// Mitsubishi GX Works2 project: PLC_GROUP_01  (1) (2)   PLC: FX3G

// global labels: Global1
VAR_GLOBAL
  DayStart AT X010 : BOOL;
  DayCoil AT Y010 : BOOL;
  DayEnd AT M0 : BOOL;
  FlourSt AT D1120 : REAL;
  FlourStock AT D1100 : REAL;
  YeastSt AT D1122 : REAL;
  YeastStock AT D1102 : REAL;
  WaterSt AT D1124 : REAL;
  WaterStock AT D1104 : REAL;
  OilSt AT D1126 : REAL;
  OilStock AT D1106 : REAL;
  SpicesSt AT D1128 : REAL;
  SpicesStock AT D1108 : REAL;
  Shutdown AT X007 : BOOL;
  InventoryDone AT M18 : BOOL;
  PrepCoil AT Y005 : BOOL;
END_VAR
VAR_GLOBAL CONSTANT
  Const_100 : REAL := 100;
  Yeast_MUL : REAL := 0.2;
END_VAR
VAR_GLOBAL
  YeastCheck AT D1130 : REAL;
END_VAR
VAR_GLOBAL CONSTANT
  Water_MUL : REAL := 0.5;
END_VAR
VAR_GLOBAL
  WaterCheck AT D1132 : REAL;
END_VAR
VAR_GLOBAL CONSTANT
  Oil_MUL : REAL := 0.3;
END_VAR
VAR_GLOBAL
  OilCheck AT D1134 : REAL;
END_VAR
VAR_GLOBAL CONSTANT
  Spices_MUL : REAL := 0.1;
END_VAR
VAR_GLOBAL
  SpicesCheck AT D1136 : REAL;
  blink2 AT M50 : BOOL;
  TS1 AT M50 : BOOL;
  blinktest AT TS1 : BOOL;
  blink3 AT M52 : BOOL;
  blinktest2 AT TS2 : BOOL;
  blinkA AT TC1 : BOOL;
END_VAR
VAR_GLOBAL CONSTANT
  blinktimems : INT := 5;
END_VAR
VAR_GLOBAL
  blinkB AT TC2 : BOOL;
  EndBlink10 AT CC1 : BOOL;
END_VAR
VAR_GLOBAL CONSTANT
  Count_10 : INT := 6;
END_VAR
VAR_GLOBAL
  EndBlink10_O AT CS1 : BOOL;
  DayCoilchecker AT M20 : BOOL;
  DayEndBlink AT M22 : BOOL;
  PrepStart AT X002 : BOOL;
  PrepT AT TC3 : BOOL;
END_VAR
VAR_GLOBAL CONSTANT
  LightT : INT := 30;
END_VAR
VAR_GLOBAL
  PrepCoilOff AT TS3 : BOOL;
END_VAR
VAR_GLOBAL CONSTANT
  Const_30 : REAL := 30;
  Const_50 : REAL := 50;
  Const_20 : REAL := 20;
  Const_10 : REAL := 10;
END_VAR
VAR_GLOBAL
  TempFlour AT D2000 : REAL;
  TempOil AT D2002 : REAL;
  TempWater AT D2004 : REAL;
  TempYeast AT D2006 : REAL;
  TempSpices AT D2008 : REAL;
  KneadStart AT X001 : BOOL;
  KneadStage AT M30 : BOOL;
  KneadCoil AT Y001 : BOOL;
  MixerStock AT D1110 : REAL;
END_VAR
VAR_GLOBAL CONSTANT
  Const_210 : REAL := 210;
END_VAR
VAR_GLOBAL
  FinishTransfer AT M4 : BOOL;
  Knead AT X011 : BOOL;
  RiseStart AT X011 : BOOL;
  RiseStage AT M40 : BOOL;
  EndBlinkRise AT CS10 : BOOL;
  EndBlinkRise1 AT CC10 : BOOL;
  blinkRise AT M41 : BOOL;
  blinkA_R AT TC10 : BOOL;
  blinkA_R1 AT TS10 : BOOL;
  blinkB_R AT TC11 : BOOL;
  Coil2 AT Y002 : BOOL;
  blinkB_R1 AT TS11 : BOOL;
  Coil3 AT Y003 : BOOL;
  RiseStorage AT D1114 : REAL;
  CountC11 AT CC20 : BOOL;
END_VAR
VAR_GLOBAL CONSTANT
  Count_2 : INT := 2;
END_VAR
VAR_GLOBAL
  CountC11End AT CS20 : BOOL;
  CountC5 AT CC5 : BOOL;
  CountC5End AT CS5 : BOOL;
  RiseSt1 AT M45 : BOOL;
  RiseEnd AT CS10 : BOOL;
  BakeStart AT M60 : BOOL;
  BakingPan AT D1118 : REAL;
  BakeT AT TC14 : BOOL;
END_VAR
VAR_GLOBAL CONSTANT
  LightBakeT : INT := 40;
END_VAR
VAR_GLOBAL
  BakeCoilOff AT TS14 : BOOL;
  BakeCoil AT Y004 : BOOL;
  QA3 AT X003 : BOOL;
END_VAR
VAR_GLOBAL CONSTANT
  Const_1 : REAL := 1;
  Const_5 : REAL := 5;
END_VAR
VAR_GLOBAL
  QA_TRUE AT M80 : BOOL;
  QA_T AT TC15 : BOOL;
END_VAR
VAR_GLOBAL CONSTANT
  LightQAT : INT := 50;
END_VAR
VAR_GLOBAL
  QA_Off AT TS15 : BOOL;
  QACoil AT Y006 : BOOL;
  Shelf AT D3333 : REAL;
  LTAnalogCheck AT M82 : BOOL;
  RST_All AT M100 : BOOL;
  Analog_Moved AT M83 : BOOL;
END_VAR
VAR_GLOBAL CONSTANT
  Const_400 : INT := 400;
  Const_2000 : INT := 2000;
END_VAR
VAR_GLOBAL
  Analog_Value AT D8490 : REAL;
  QA_TRUE2 AT M83 : BOOL;
  Analog_Input_2 AT D8281 : INT;
  RiseMoved AT M61 : BOOL;
  Coil4ON AT M61 : BOOL;
  FlourDone AT M19 : BOOL;
END_VAR

// task Task_01 (event TRUE, interval 0, priority 31): POU_01

PROGRAM POU_01
(* structured ladder/FBD written out as ST: instructions are called as NAME(EN, inputs, outputs); _pN, _eN, _tN stand for wires *)
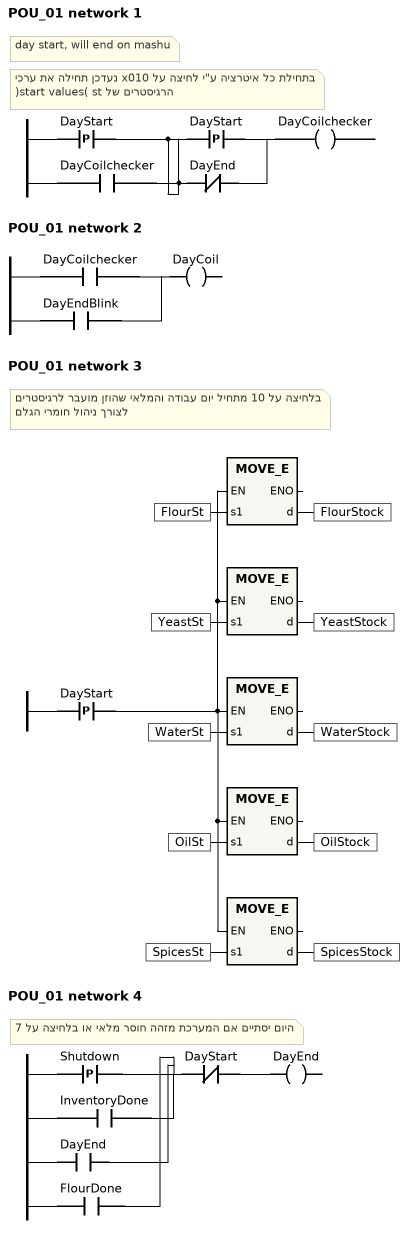
(* network 1 *)
(* day start, will end on mashu *)
(* בתחילת כל איטרציה ע"י לחיצה על x010 נעדכן תחילה את ערכי הרגיסטרים של st )start values( *)
_p1 := LDP(TRUE, DayStart) OR DayCoilchecker;
DayCoilchecker := (_p1 AND LDP(TRUE, DayStart)) OR (_p1 AND NOT DayEnd);
(* network 2 *)
DayCoil := DayCoilchecker OR DayEndBlink;
(* network 3 *)
(* בלחיצה על 10 מתחיל יום עבודה והמלאי שהוזן מועבר לרגיסטרים לצורך ניהול חומרי הגלם *)
_p1 := LDP(TRUE, DayStart);
MOVE_E(_p1, FlourSt, FlourStock);
MOVE_E(_p1, YeastSt, YeastStock);
MOVE_E(_p1, WaterSt, WaterStock);
MOVE_E(_p1, OilSt, OilStock);
MOVE_E(_p1, SpicesSt, SpicesStock);
(* network 4 *)
(* היום יסתיים אם המערכת מזהה חוסר מלאי או בלחיצה על 7 *)
DayEnd := (LDP(TRUE, Shutdown) OR InventoryDone OR DayEnd OR FlourDone) AND NOT DayStart;
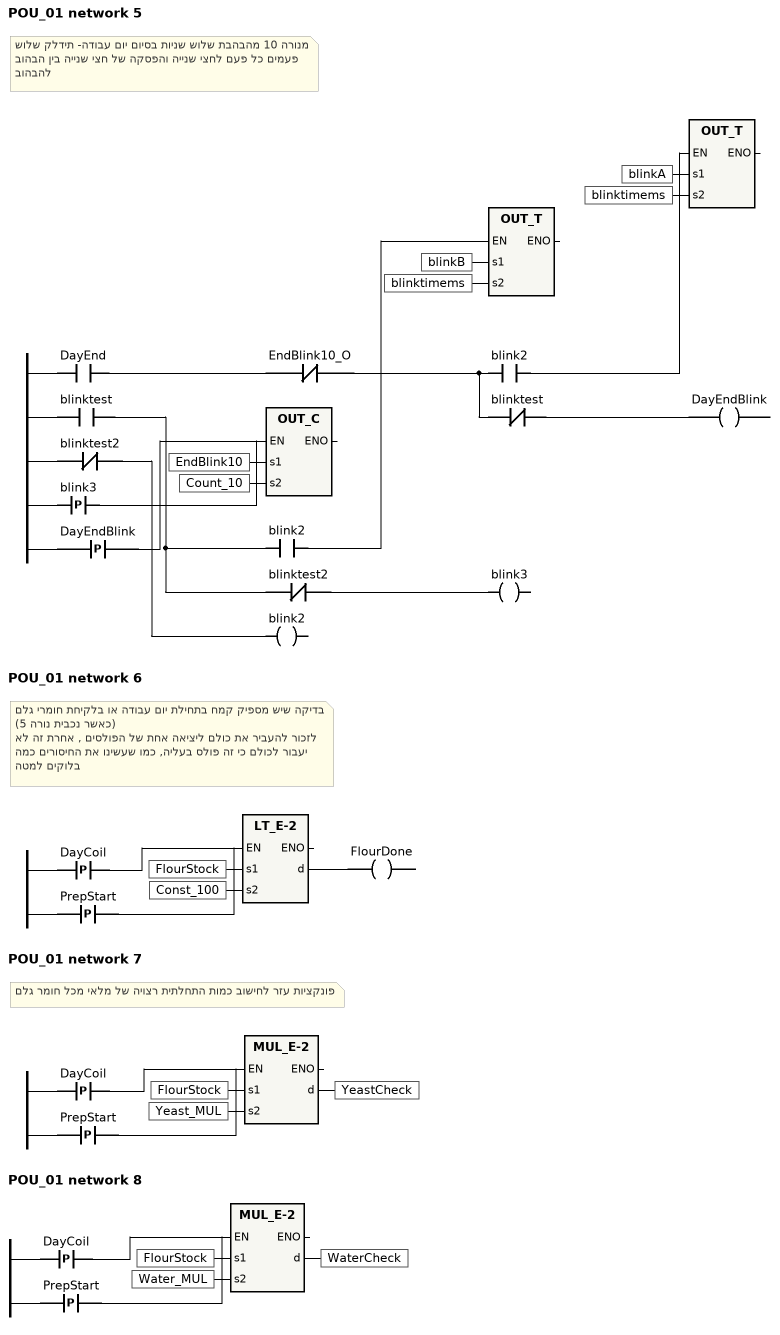
(* network 5 *)
(* מנורה 10 מהבהבת שלוש שניות בסיום יום עבודה- תידלק שלוש פעמים כל פעם לחצי שנייה והפסקה של חצי שנייה בין הבהוב להבהוב *)
_p1 := DayEnd AND NOT EndBlink10_O;
OUT_T(_p1 AND blink2, blinkA, blinktimems);
DayEndBlink := _p1 AND NOT blinktest;
OUT_T(blinktest AND blink2, blinkB, blinktimems);
blink3 := blinktest AND NOT blinktest2;
blink2 := NOT blinktest2;
OUT_C(LDP(TRUE, blink3) OR LDP(TRUE, DayEndBlink), EndBlink10, Count_10);
(* network 6 *)
(* בדיקה שיש מספיק קמח בתחילת יום עבודה או בלקיחת חומרי גלם (כאשר נכבית נורה 5)                                                            לזכור להעביר את כולם ליציאה אחת של הפולסים , אחרת זה לא יעבור לכולם כי זה פולס בעליה, כמו שעשינו את החיסורים כמה בלוקים למטה *)
LT_E(LDP(TRUE, DayCoil) OR LDP(TRUE, PrepStart), FlourStock, Const_100, _t1);
FlourDone := _t1;
(* network 7 *)
(* פונקציות עזר לחישוב כמות התחלתית רצויה של מלאי מכל חומר גלם *)
MUL_E(LDP(TRUE, DayCoil) OR LDP(TRUE, PrepStart), FlourStock, Yeast_MUL, YeastCheck);
(* network 8 *)
MUL_E(LDP(TRUE, DayCoil) OR LDP(TRUE, PrepStart), FlourStock, Water_MUL, WaterCheck);
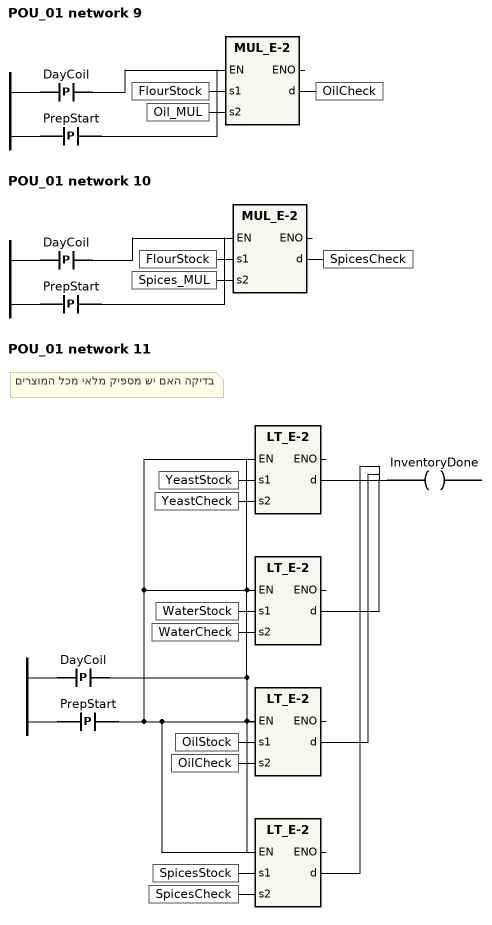
(* network 9 *)
MUL_E(LDP(TRUE, DayCoil) OR LDP(TRUE, PrepStart), FlourStock, Oil_MUL, OilCheck);
(* network 10 *)
MUL_E(LDP(TRUE, DayCoil) OR LDP(TRUE, PrepStart), FlourStock, Spices_MUL, SpicesCheck);
(* network 11 *)
(* בדיקה האם יש מספיק מלאי מכל המוצרים *)
_p1 := LDP(TRUE, DayCoil) OR LDP(TRUE, PrepStart);
LT_E(_p1, YeastStock, YeastCheck, _t2);
LT_E(_p1, WaterStock, WaterCheck, _t3);
LT_E(_p1, OilStock, OilCheck, _t4);
LT_E(_p1, SpicesStock, SpicesCheck, _t5);
InventoryDone := _t2 OR _t3 OR _t4 OR _t5;
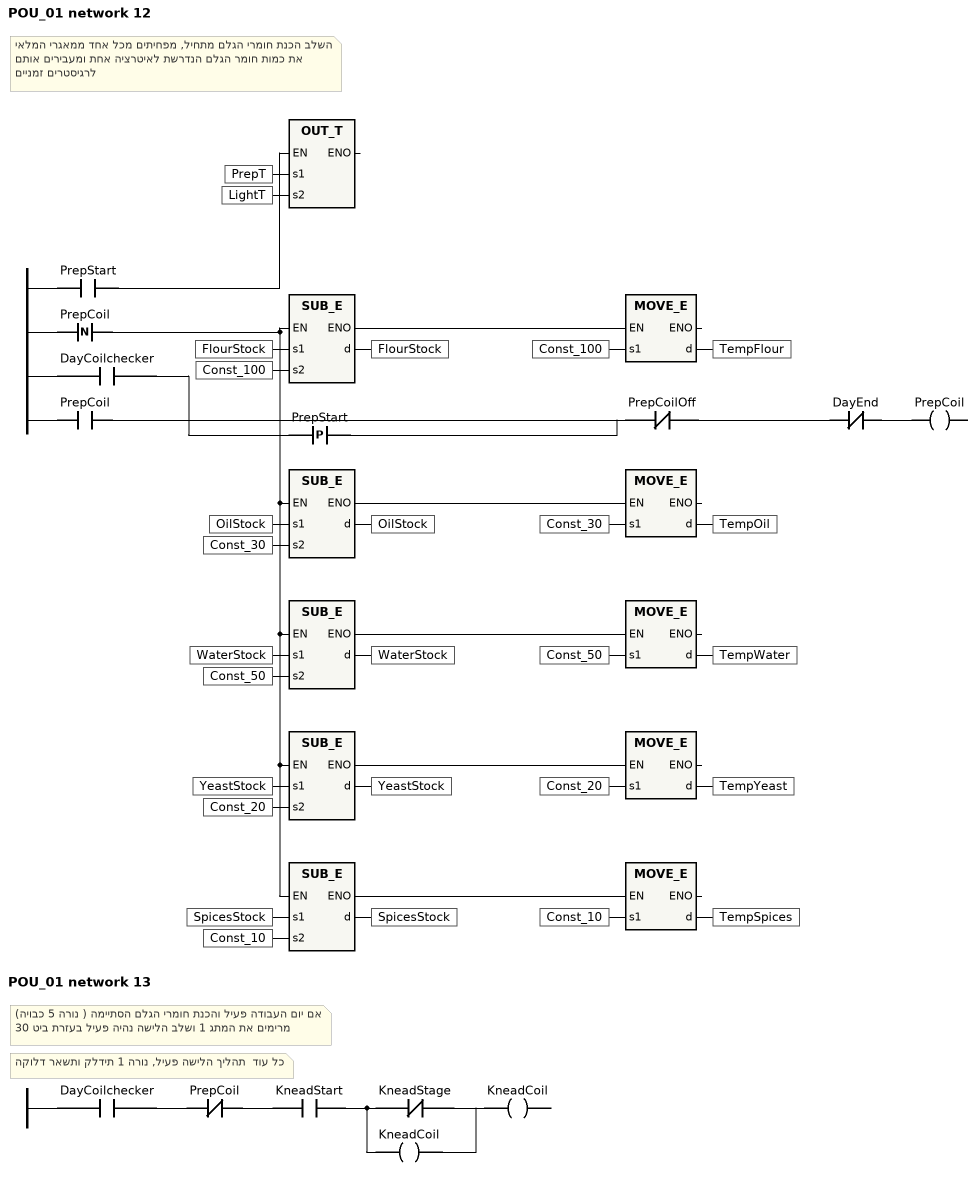
(* network 12 *)
(* השלב הכנת חומרי הגלם מתחיל, מפחיתים מכל אחד ממאגרי המלאי את כמות חומר הגלם הנדרשת לאיטרציה אחת ומעבירים אותם לרגיסטרים זמניים *)
OUT_T(PrepStart, PrepT, LightT);
_p1 := LDF(TRUE, PrepCoil);
_e2 := SUB_E(_p1, FlourStock, Const_100, FlourStock);
MOVE_E(_e2, Const_100, TempFlour);
_e3 := SUB_E(_p1, OilStock, Const_30, OilStock);
MOVE_E(_e3, Const_30, TempOil);
_e4 := SUB_E(_p1, WaterStock, Const_50, WaterStock);
MOVE_E(_e4, Const_50, TempWater);
_e5 := SUB_E(_p1, YeastStock, Const_20, YeastStock);
MOVE_E(_e5, Const_20, TempYeast);
_e6 := SUB_E(_p1, SpicesStock, Const_10, SpicesStock);
MOVE_E(_e6, Const_10, TempSpices);
PrepCoil := (((DayCoilchecker AND LDP(TRUE, PrepStart)) OR PrepCoil) AND NOT PrepCoilOff) AND NOT DayEnd;
(* network 13 *)
(* אם יום העבודה פעיל והכנת חומרי הגלם הסתיימה ( נורה 5 כבויה) מרימים את המתג 1 ושלב הלישה נהיה פעיל בעזרת ביט 30 *)
(* כל עוד  תהליך הלישה פעיל, נורה 1 תידלק ותשאר דלוקה *)
_p1 := DayCoilchecker AND NOT PrepCoil AND KneadStart;
KneadCoil := _p1;
KneadCoil := (_p1 AND NOT KneadStage) OR _p1;
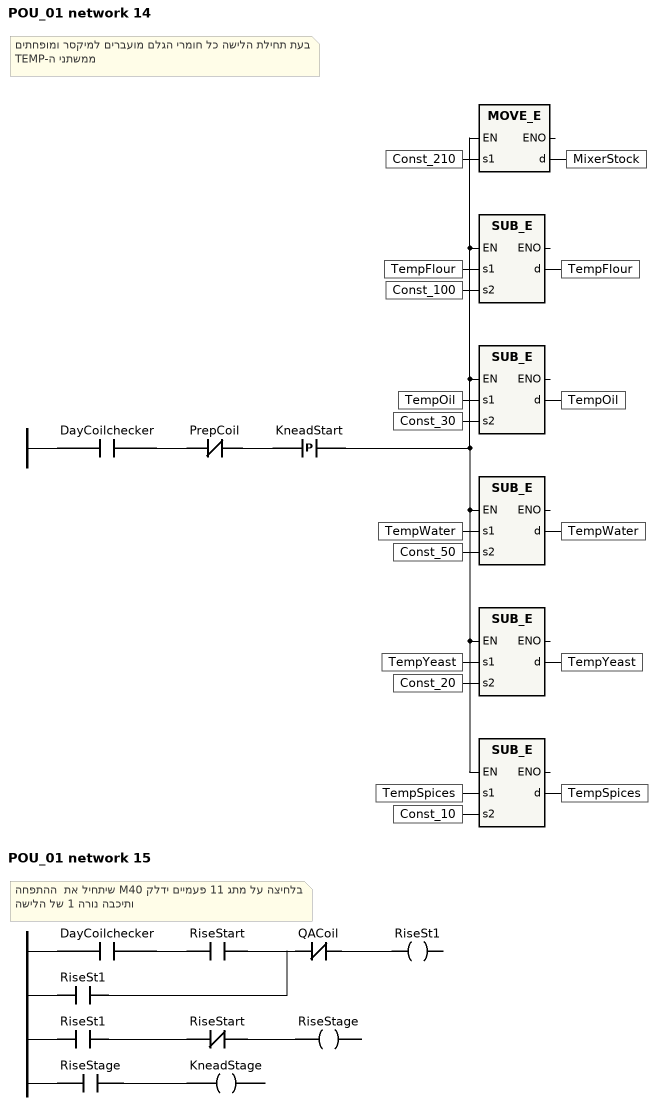
(* network 14 *)
(* בעת תחילת הלישה כל חומרי הגלם מועברים למיקסר ומופחתים ממשתני ה-TEMP *)
_p1 := DayCoilchecker AND NOT PrepCoil AND LDP(TRUE, KneadStart);
MOVE_E(_p1, Const_210, MixerStock);
SUB_E(_p1, TempFlour, Const_100, TempFlour);
SUB_E(_p1, TempOil, Const_30, TempOil);
SUB_E(_p1, TempWater, Const_50, TempWater);
SUB_E(_p1, TempYeast, Const_20, TempYeast);
SUB_E(_p1, TempSpices, Const_10, TempSpices);
(* network 15 *)
(* בלחיצה על מתג 11 פעמיים ידלק M40 שיתחיל את  ההתפחה ותיכבה נורה 1 של הלישה *)
RiseSt1 := ((DayCoilchecker AND RiseStart) OR RiseSt1) AND NOT QACoil;
RiseStage := RiseSt1 AND NOT RiseStart;
KneadStage := RiseStage;
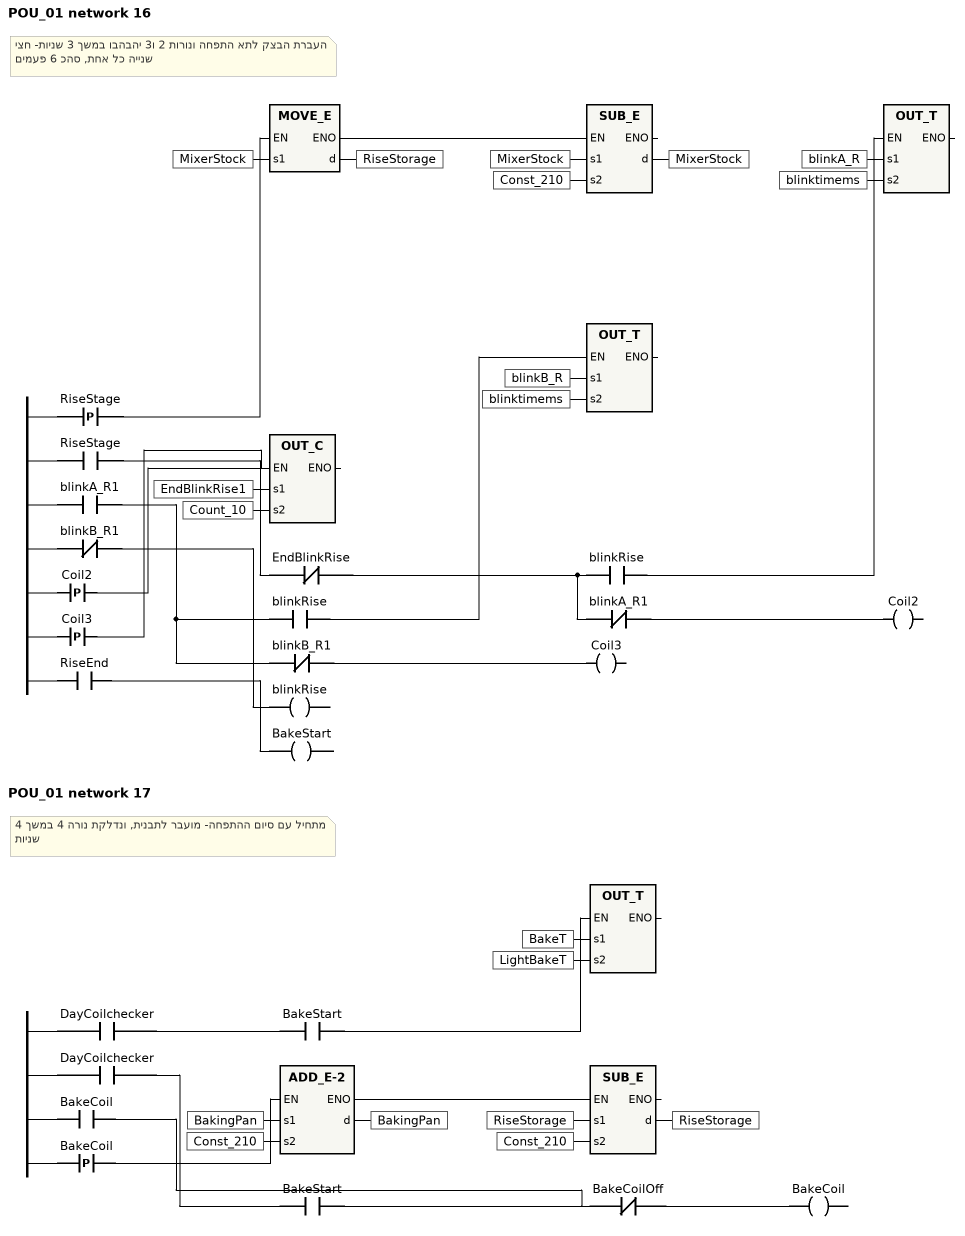
(* network 16 *)
(* העברת הבצק לתא התפחה ונורות 2 ו3 יהבהבו במשך 3 שניות- חצי שנייה כל אחת, סהכ 6 פעמים *)
_e1 := MOVE_E(LDP(TRUE, RiseStage), MixerStock, RiseStorage);
SUB_E(_e1, MixerStock, Const_210, MixerStock);
_p2 := RiseStage AND NOT EndBlinkRise;
OUT_T(_p2 AND blinkRise, blinkA_R, blinktimems);
Coil2 := _p2 AND NOT blinkA_R1;
OUT_T(blinkA_R1 AND blinkRise, blinkB_R, blinktimems);
Coil3 := blinkA_R1 AND NOT blinkB_R1;
blinkRise := NOT blinkB_R1;
OUT_C(LDP(TRUE, Coil2) OR LDP(TRUE, Coil3), EndBlinkRise1, Count_10);
BakeStart := RiseEnd;
(* network 17 *)
(* מתחיל עם סיום ההתפחה- מועבר לתבנית, ונדלקת נורה 4 במשך 4 שניות *)
OUT_T(DayCoilchecker AND BakeStart, BakeT, LightBakeT);
BakeCoil := ((DayCoilchecker AND BakeStart) OR BakeCoil) AND NOT BakeCoilOff;
_e1 := ADD_E(LDP(TRUE, BakeCoil), BakingPan, Const_210, BakingPan);
SUB_E(_e1, RiseStorage, Const_210, RiseStorage);
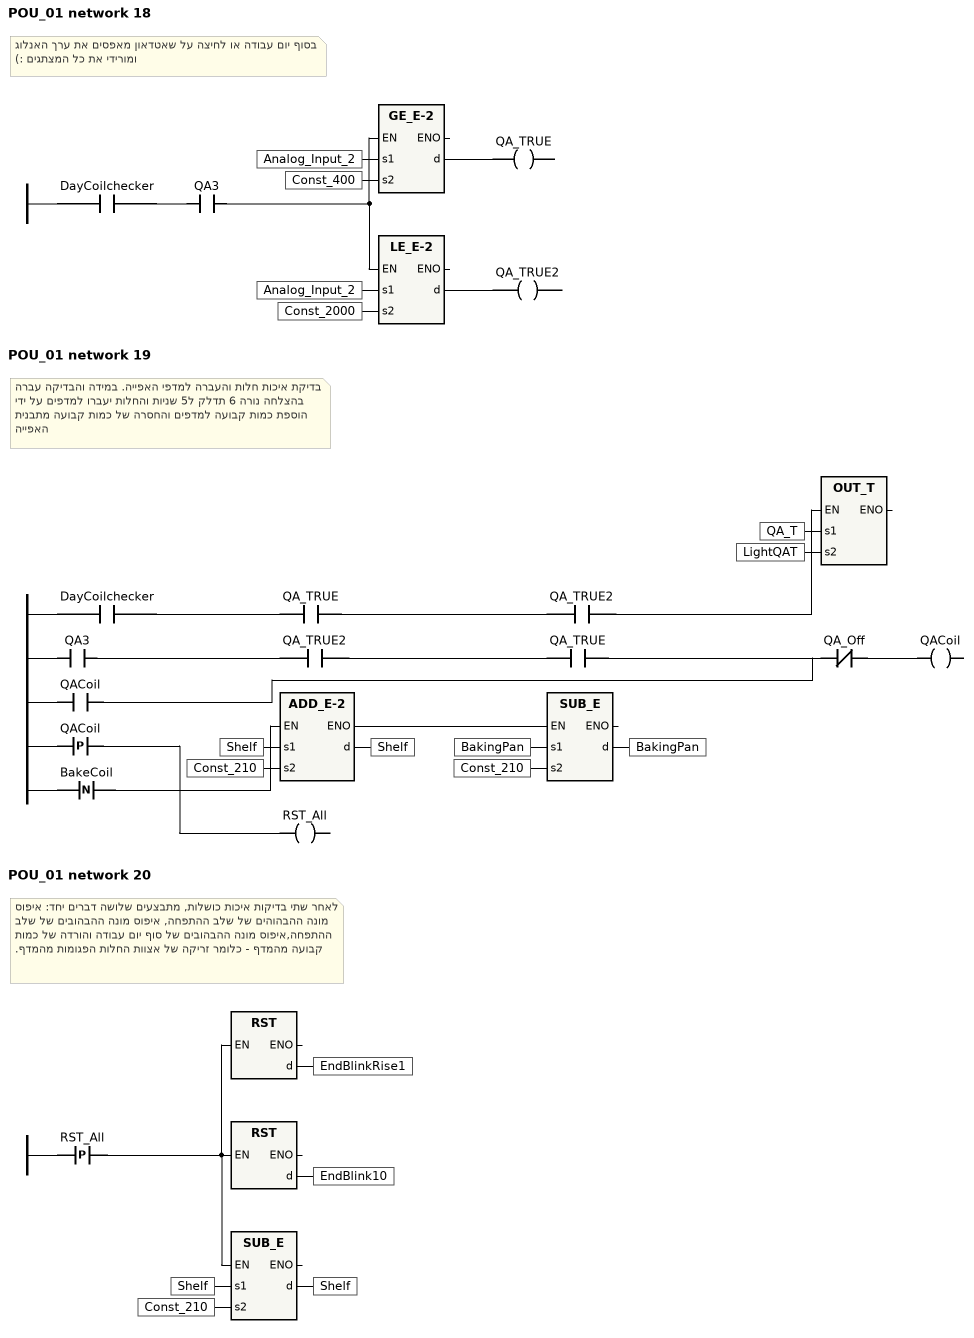
(* network 18 *)
(* בסוף יום עבודה או לחיצה על שאטדאון מאפסים את ערך האנלוג ומורידי את כל המצתגים :) *)
_p1 := DayCoilchecker AND QA3;
GE_E(_p1, Analog_Input_2, Const_400, _t2);
QA_TRUE := _t2;
LE_E(_p1, Analog_Input_2, Const_2000, _t3);
QA_TRUE2 := _t3;
(* network 19 *)
(* בדיקת איכות חלות והעברה למדפי האפייה. במידה והבדיקה עברה בהצלחה נורה 6 תדלק ל5 שניות והחלות יעברו למדפים על ידי הוספת כמות קבועה למדפים והחסרה של כמות קבועה מתבנית האפייה *)
OUT_T(DayCoilchecker AND QA_TRUE AND QA_TRUE2, QA_T, LightQAT);
QACoil := ((QA3 AND QA_TRUE2 AND QA_TRUE) OR QACoil) AND NOT QA_Off;
RST_All := LDP(TRUE, QACoil);
_e1 := ADD_E(LDF(TRUE, BakeCoil), Shelf, Const_210, Shelf);
SUB_E(_e1, BakingPan, Const_210, BakingPan);
(* network 20 *)
(* לאחר שתי בדיקות איכות כושלות, מתבצעים שלושה דברים יחד: איפוס מונה ההבהוהים של שלב ההתפחה, איפוס מונה ההבהובים של שלב ההתפחה,איפוס מונה ההבהובים של סוף יום עבודה והורדה של כמות קבועה מהמדף - כלומר זריקה של אצוות החלות הפגומות מהמדף. *)
_p1 := LDP(TRUE, RST_All);
RST(_p1, EndBlinkRise1);
RST(_p1, EndBlink10);
SUB_E(_p1, Shelf, Const_210, Shelf);
END_PROGRAM
